ADAPTER ACylinder
  (* Standard: 61499-1 *)
  (* Version 0.0, 2008-04-22, GE, 4DIAC-Consortium *)
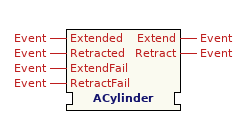
  EVENT_INPUT
    Extended; (* Response from Socket *)
    Retracted; (* Response from Socket *)
    ExtendFail;
    RetractFail;
  END_EVENT
  EVENT_OUTPUT
    Extend;
    Retract;
  END_EVENT
  SERVICE PLUG/SOCKET
    SEQUENCE ExtendSuccess
      PLUG.Extend() -> SOCKET.Extend(REQD);
      SOCKET.StatusExtend(CNFD) -> PLUG.StatusExtend(CNFD);
    END_SEQUENCE
    SEQUENCE RetractSuccess
      PLUG.Retract() -> SOCKET.Retract();
      SOCKET.StatusRetract() -> PLUG.StatusRetract();
    END_SEQUENCE
    SEQUENCE ExtendFail
      PLUG.Extend() -> SOCKET.Extend();
      SOCKET.ExtendFail() -> PLUG.ExtendFail();
    END_SEQUENCE
    SEQUENCE RetarctFail
      PLUG.Retract() -> SOCKET.Retract();
      SOCKET.RetractFail() -> PLUG.RetractFail();
    END_SEQUENCE
  END_SERVICE
END_ADAPTER
